// Mitsubishi GX Works2 project: inc_decEx01   PLC: Q02/Q02H

PROGRAM MAIN
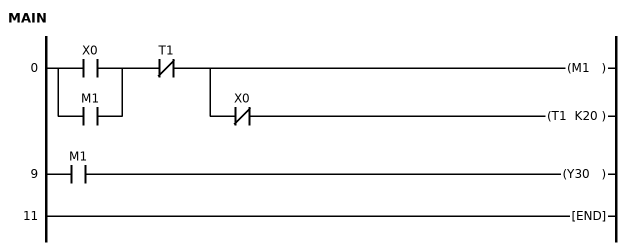
0     LD      X0
      OR      M1
      ANI     T1
      OUT     M1
      ANI     X0
      OUT     T1 K20
9     LD      M1
      OUT     Y30
11    END
END_PROGRAM
